Staubli VAL3: new.pgx

public program new(string x_sName (dimensions=1), num& x_nResult[] (dimensions=1))
  local string l_sMessage
begin
  // new element
  if insert(saveProg:pProg[x_sName])
    saveProg:pProg[x_sName].sID=x_sName
    x_nResult=0
  else
    call language:message(l_sMessage,-2)
    popUpMsg(l_sMessage)
    x_nResult=-1
  endIf
end
